KUKA KRL data list: getBlockBase.dat

&ACCESS RVO
&REL 6
DEFDAT getBlockBase PUBLIC

ENDDAT
